// TwinCAT 3 PLC project TcoDrivesBeckhoffTests
// Title: TcoDrivesBeckhoffTests
// Company: Vortex.Library
// Author: TcOpenGroup
// ProjectVersion: 0.6.0.913
// ProgramVersion: 3.1.4026.12
// libraries:
//   Tc2_EtherCAT, * (Beckhoff Automation GmbH)
//   Tc2_MC2, * (Beckhoff Automation GmbH)
//   Tc2_Standard, * (Beckhoff Automation GmbH)
//   Tc2_System, * (Beckhoff Automation GmbH)
//   Tc3_Module, * (Beckhoff Automation GmbH)
//   TcoCore, 0.6.0.913 (Vortex.Library)
//   TcoDrivesBeckhoff, 0.6.0.913 (Vortex.Library)
// project tree:
//   GVLs/ GVL.TcGVL (not stored)
//   / PlcTask1.TcTTO (not stored)
//   POUs/ MAIN.TcPOU (not stored)
//   Tests/TcoContext/ Sequence1Task.TcPOU (not stored), SomeTestPositions.TcPOU (not stored), SomeTestMultiPositions.TcPOU, WpfContext.TcPOU (not stored)
//   Tests/TcoContext/WrappedComponent/ WrappedComponentExample.TcPOU (not stored), WrappedComponentExample_Config.TcDUT (not stored), WrappedComponentExample_Control.TcDUT (not stored), WrappedComponentExample_Status.TcDUT (not stored), WrappedComponentsExample.TcDUT (not stored)
//   Tests/TcoDriveSimple/ eTcoDriveSimpleTests.TcDUT (not stored), TcoDriveSimpleTestContext.TcPOU (not stored), TcoDriveSimpleTest.TcPOU (not stored)
//   Tests/TcoSingleAxis/ eTcoSingleAxisTests.TcDUT (not stored), TcoSingleAxisContext.TcPOU (not stored), TcoSingleAxisTest.TcPOU (not stored)
//   Tests/TcoMultiAxis/ eTcoMultiAxisTests.TcDUT (not stored), TcoMultiAxisContext.TcPOU (not stored), TcoMultiAxisTest.TcPOU (not stored)
// (motion and I/O tree: see PLC project tcodrivesbeckhoff)
// real-time tasks:
//   TASK PlcTask: cycle T#10ms, priority 20, ADS port 350
//   TASK PlcTask1: cycle T#10ms, priority 1, ADS port 351
// variable links:
//   TcoDrivesBeckhoffTests/TcoDrivesBeckhoffTests Instance <-> Device 2 (EtherCAT)/Term 1 (EK1200)/Term 12 (EL1809)
//     PlcTask1 Inputs/GVL._calibrationCam <-> Channel 1/Input
//   TcoDrivesBeckhoffTests/TcoDrivesBeckhoffTests Instance <-> NC-Task 1 SAF/Axes/Axis 1
//     PlcTask1 Inputs/GVL.Axis1.NcToPlc <-> Outputs/ToPlc
//     PlcTask1 Outputs/GVL.Axis1.PlcToNc <-> Inputs/FromPlc
//   TcoDrivesBeckhoffTests/TcoDrivesBeckhoffTests Instance <-> NC-Task 1 SAF/Axes/Axis 2
//     PlcTask1 Inputs/GVL.Axis2.NcToPlc <-> Outputs/ToPlc
//     PlcTask1 Outputs/GVL.Axis2.PlcToNc <-> Inputs/FromPlc
//   TcoDrivesBeckhoffTests/TcoDrivesBeckhoffTests Instance <-> NC-Task 1 SAF/Axes/Axis 3
//     PlcTask1 Inputs/GVL.Axis3.NcToPlc <-> Outputs/ToPlc
//     PlcTask1 Outputs/GVL.Axis3.PlcToNc <-> Inputs/FromPlc
//   TcoDrivesBeckhoffTests/TcoDrivesBeckhoffTests Instance <-> NC-Task 1 SAF/Axes/Axis 4
//     PlcTask1 Inputs/GVL.Axis4.NcToPlc <-> Outputs/ToPlc
//     PlcTask1 Outputs/GVL.Axis4.PlcToNc <-> Inputs/FromPlc

// ---- Tests/TcoContext/SomeTestMultiPositions.TcPOU
FUNCTION_BLOCK SomeTestMultiPositions EXTENDS TcoDrivesBeckhoff.TcoMultiAxisPositionsRootContainer
VAR_INPUT
END_VAR
VAR_OUTPUT
END_VAR
VAR
	{attribute addProperty Name "<#Pick Position#>"}
	PickPosition:TcoDrivesBeckhoff.TcoMultiAxisMoveParam;
	{attribute addProperty Name "<#Place  Position#>"}
	PlacePosition:TcoDrivesBeckhoff.TcoMultiAxisMoveParam;

END_VAR

PROPERTY PUBLIC PickPos : REFERENCE TO TcoDrivesBeckhoff.TcoMultiAxisMoveParam;
GET
PickPos REF=PickPosition;
END_GET
END_PROPERTY

PROPERTY PUBLIC PlacePos : REFERENCE TO TcoDrivesBeckhoff.TcoMultiAxisMoveParam;
GET
PlacePos REF=PlacePosition;
END_GET
END_PROPERTY

END_FUNCTION_BLOCK
